Fanuc KAREL source: kb00062.KL

PROGRAM KB00062
%STACKSIZE=65535
%PRIORITY=65535
%NOLOCKGROUP
VAR
P1 : INTEGER
P3 : ARRAY[4] OF INTEGER
P4 : INTEGER
-- UNRESOLVED DECLARATIONS (source type spelling not recovered)
-- P2 : TYPE_0x1100 (type_u16=0x1100)
BEGIN
P1=1
P3[1]=1
P4=1
DELETE_QUEUE(P1,P2,P3,P4)
END KB00062
